TYPE DUT :
STRUCT
	Encoder:LREAL;
	LeftTop:LREAL;
END_STRUCT
END_TYPE

(* stored: Version 1.1.0.1, ProductVersion 3.1.4024.6
   DUT DUT: Id {c1a16892-445a-4feb-8da5-94fd732edf37} *)
